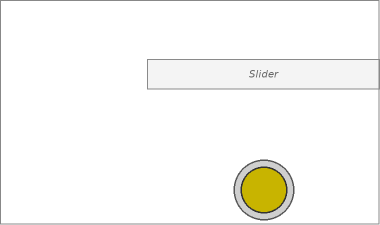
VISUALIZATION Visualization  // 380x225
    Lamp1 (229,155 70x70), variable: GVL.lightStatus, style: Lamp-Lamp1-Yellow
    Slider (147,59 233x30), variable: GVL.distance, scale 0..5
END_VISUALIZATION

(* stored: Version 1.1.0.1, ProductVersion 3.1.4024.12
   Visu Visualization: Id {9bab2fdf-fe47-4714-9cce-5c090549dde9} *)
